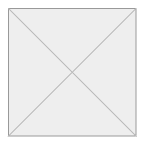
[picture p24: Yellow_Ind (HMI screen)]
bitmap at (0,0)-(128,128): c:\flexlink\bitmap\button_blank_gray_01.bmp
bitmap at (0,0)-(128,128): c:\flexlink\bitmap\button_blank_yellow_01.bmp
*)
